FUNCTION_BLOCK Room_Ctx
VAR_INPUT
	io		: Room_Ctx_Io;
	hmi		: Room_Ctx_Hmi;
	state	: Room_Ctx_States;
	priv	: Room_Ctx_Priv;
END_VAR

END_FUNCTION_BLOCK

(* stored: Version 1.1.0.1
   POU Room_Ctx: Id {8aac3efc-2438-43bb-b2e7-024ad5e5c587}, SpecialFunc None *)
